{attribute 'qualified_only'}
{attribute 'strict'}
TYPE E_ActivePopup :
(
    NONE            := 0,
    PUCK_REMOVAL    := 1,
    REJECT_PART     := 2,
    DISABLED_NEST   := 3,
    REJECT_BIN_FULL := 4
);
END_TYPE

(* stored: Version 1.1.0.1
   DUT E_ActivePopup: Id {694504d3-b6cf-430f-8d6d-bf46a3dc3589} *)
